(* IEC 61131-3 sources: sF/scufford/src/typeLib/modules/STBlocks, 1 file *)

(* ---- sinST.st ---- *)
PROGRAM execute
VAR
    input1: REAL;
    output1: REAL;
END_VAR

output1 := SIN(input1);
END_PROGRAM
